PROGRAM TestAblauf
VAR
END_VAR

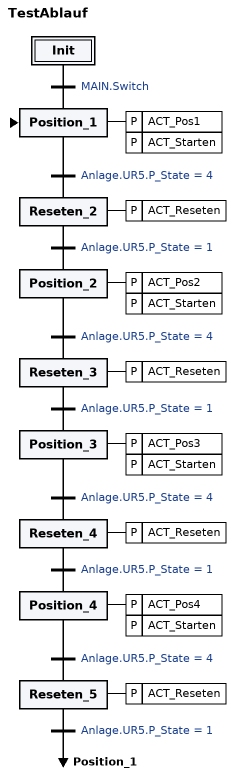
INITIAL_STEP Init:
END_STEP
TRANSITION FROM Init TO Position_1
    := MAIN.Switch;
END_TRANSITION
STEP Position_1:
    ACT_Pos1(P);
    ACT_Starten(P);
END_STEP
TRANSITION FROM Position_1 TO Reseten_2
    := Anlage.UR5.P_State = 4;
END_TRANSITION
STEP Reseten_2:
    ACT_Reseten(P);
END_STEP
TRANSITION FROM Reseten_2 TO Position_2
    := Anlage.UR5.P_State = 1;
END_TRANSITION
STEP Position_2:
    ACT_Pos2(P);
    ACT_Starten(P);
END_STEP
TRANSITION FROM Position_2 TO Reseten_3
    := Anlage.UR5.P_State = 4;
END_TRANSITION
STEP Reseten_3:
    ACT_Reseten(P);
END_STEP
TRANSITION FROM Reseten_3 TO Position_3
    := Anlage.UR5.P_State = 1;
END_TRANSITION
STEP Position_3:
    ACT_Pos3(P);
    ACT_Starten(P);
END_STEP
TRANSITION FROM Position_3 TO Reseten_4
    := Anlage.UR5.P_State = 4;
END_TRANSITION
STEP Reseten_4:
    ACT_Reseten(P);
END_STEP
TRANSITION FROM Reseten_4 TO Position_4
    := Anlage.UR5.P_State = 1;
END_TRANSITION
STEP Position_4:
    ACT_Pos4(P);
    ACT_Starten(P);
END_STEP
TRANSITION FROM Position_4 TO Reseten_5
    := Anlage.UR5.P_State = 4;
END_TRANSITION
STEP Reseten_5:
    ACT_Reseten(P);
END_STEP
TRANSITION FROM Reseten_5 TO Position_1
    := Anlage.UR5.P_State = 1;
END_TRANSITION

ACTION ACT_Pos1:
MAIN.testProcessValue.q1 := 0.2;
MAIN.testProcessValue.q2 := 0;
MAIN.testProcessValue.q3 := 0;
MAIN.testProcessValue.q4 := 0;
MAIN.testProcessValue.q5 := 0;
MAIN.testProcessValue.q6 := 0;
MAIN.testProcessValue.a := 0.2;
MAIN.testProcessValue.v := 0.2;
MAIN.testProcessValue.MoveTyp := 0;
MAIN.testProcessValue.PosTyp := 1;
END_ACTION

ACTION ACT_Pos2:
MAIN.testProcessValue.q1 := 0;
MAIN.testProcessValue.q2 := 0.2;
MAIN.testProcessValue.q3 := 0;
MAIN.testProcessValue.q4 := 0;
MAIN.testProcessValue.q5 := 0;
MAIN.testProcessValue.q6 := 0;
MAIN.testProcessValue.a := 0.2;
MAIN.testProcessValue.v := 0.2;
MAIN.testProcessValue.MoveTyp := 0;
MAIN.testProcessValue.PosTyp := 1;
END_ACTION

ACTION ACT_Pos3:
MAIN.testProcessValue.q1 := -0.2;
MAIN.testProcessValue.q2 := 0;
MAIN.testProcessValue.q3 := 0;
MAIN.testProcessValue.q4 := 0;
MAIN.testProcessValue.q5 := 0;
MAIN.testProcessValue.q6 := 0;
MAIN.testProcessValue.a := 0.2;
MAIN.testProcessValue.v := 0.2;
MAIN.testProcessValue.MoveTyp := 0;
MAIN.testProcessValue.PosTyp := 1;
END_ACTION

ACTION ACT_Pos4:
MAIN.testProcessValue.q1 := 0;
MAIN.testProcessValue.q2 := -0.2;
MAIN.testProcessValue.q3 := 0;
MAIN.testProcessValue.q4 := 0;
MAIN.testProcessValue.q5 := 0;
MAIN.testProcessValue.q6 := 0;
MAIN.testProcessValue.a := 0.2;
MAIN.testProcessValue.v := 0.2;
MAIN.testProcessValue.MoveTyp := 0;
MAIN.testProcessValue.PosTyp := 1;
END_ACTION

ACTION ACT_Reseten:
MAIN.SkillCommand := 3;
END_ACTION

ACTION ACT_Starten:
MAIN.SkillCommand := 1;
END_ACTION

END_PROGRAM

(* stored: Version 1.1.0.1
   POU TestAblauf: Id {625795d4-ad61-4554-b213-7fa4fe45f675}, SpecialFunc None
   Folder 01_Positionen: Id {d53a9dd3-59c9-44cd-95e7-31cc0aad0213}
   Action ACT_Pos1: Id {922e04d0-2312-4358-b4c5-acafa539be66}
   Action ACT_Pos2: Id {fd0e0a1c-48cf-4caa-9366-93b3146a0437}
   Action ACT_Pos3: Id {d5d677c4-219d-41ee-a870-d7c643ba965b}
   Action ACT_Pos4: Id {e2599f45-11c0-46d6-9392-2cb71db80068}
   Action ACT_Reseten: Id {11cb4250-c209-4a89-afab-579d12c0d868}
   Action ACT_Starten: Id {3b0b8def-e292-4607-a614-44e840be8aeb} *)
